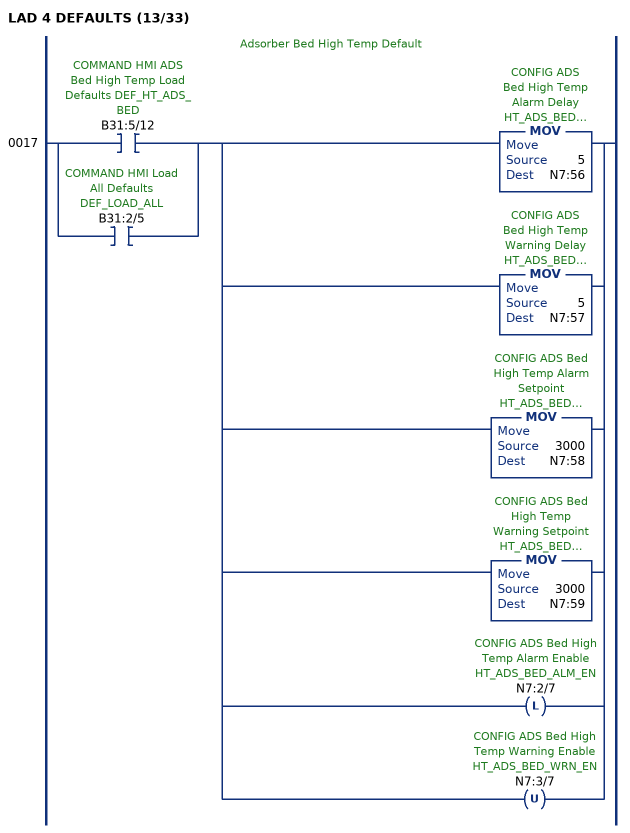
% Rung: 17 %
% Adsorber Bed High Temp Default %
SOR BST XIC B31:5/12 NXB XIC B31:2/5 BND BST MOV 5 N7:56 NXB MOV 5 N7:57 NXB MOV 3000 N7:58 NXB MOV 3000 N7:59 NXB OTL N7:2/7 NXB OTU N7:3/7 BND EOR
%   B31:5/12  DEF_HT_ADS_BED  "COMMAND HMI ADS Bed High Temp Load Defaults" %
%   B31:2/5  DEF_LOAD_ALL  "COMMAND HMI Load All Defaults" %
%   N7:56  HT_ADS_BED_ALM_DLY  "CONFIG ADS Bed High Temp Alarm Delay" %
%   N7:57  HT_ADS_BED_WRN_DLY  "CONFIG ADS Bed High Temp Warning Delay" %
%   N7:58  HT_ADS_BED_ALM_SP  "CONFIG ADS Bed High Temp Alarm Setpoint" %
%   N7:59  HT_ADS_BED_WRN_SP  "CONFIG ADS Bed High Temp Warning Setpoint" %
%   N7:2/7  HT_ADS_BED_ALM_EN  "CONFIG ADS Bed High Temp Alarm Enable" %
%   N7:3/7  HT_ADS_BED_WRN_EN  "CONFIG ADS Bed High Temp Warning Enable" %

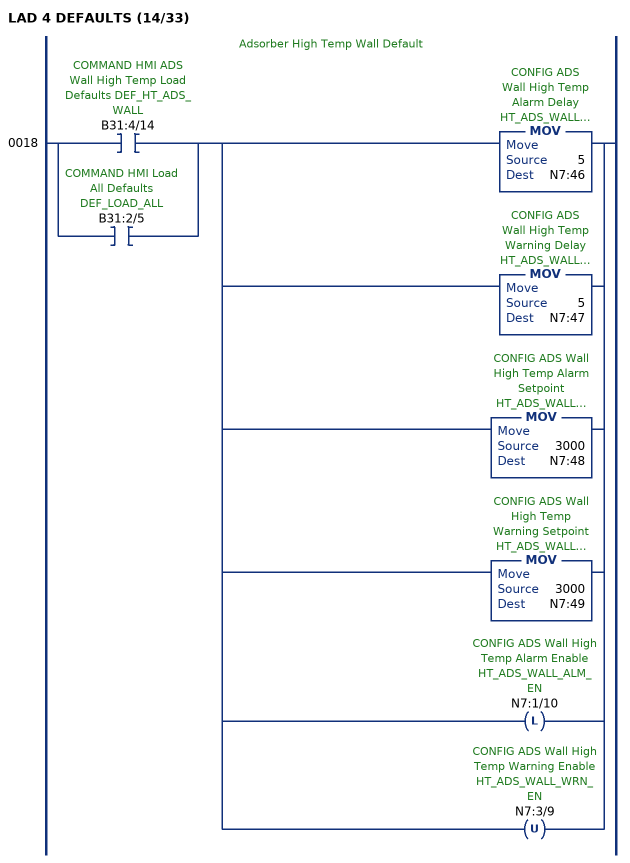
% Rung: 18 %
% Adsorber High Temp Wall Default %
SOR BST XIC B31:4/14 NXB XIC B31:2/5 BND BST MOV 5 N7:46 NXB MOV 5 N7:47 NXB MOV 3000 N7:48 NXB MOV 3000 N7:49 NXB OTL N7:1/10 NXB OTU N7:3/9 BND EOR
%   B31:4/14  DEF_HT_ADS_WALL  "COMMAND HMI ADS Wall High Temp Load Defaults" %
%   B31:2/5  DEF_LOAD_ALL  "COMMAND HMI Load All Defaults" %
%   N7:46  HT_ADS_WALL_ALM_DLY  "CONFIG ADS Wall High Temp Alarm Delay" %
%   N7:47  HT_ADS_WALL_WRN_DLY  "CONFIG ADS Wall High Temp Warning Delay" %
%   N7:48  HT_ADS_WALL_ALM_SP  "CONFIG ADS Wall High Temp Alarm Setpoint" %
%   N7:49  HT_ADS_WALL_WRN_SP  "CONFIG ADS Wall High Temp Warning Setpoint" %
%   N7:1/10  HT_ADS_WALL_ALM_EN  "CONFIG ADS Wall High Temp Alarm Enable" %
%   N7:3/9  HT_ADS_WALL_WRN_EN  "CONFIG ADS Wall High Temp Warning Enable" %

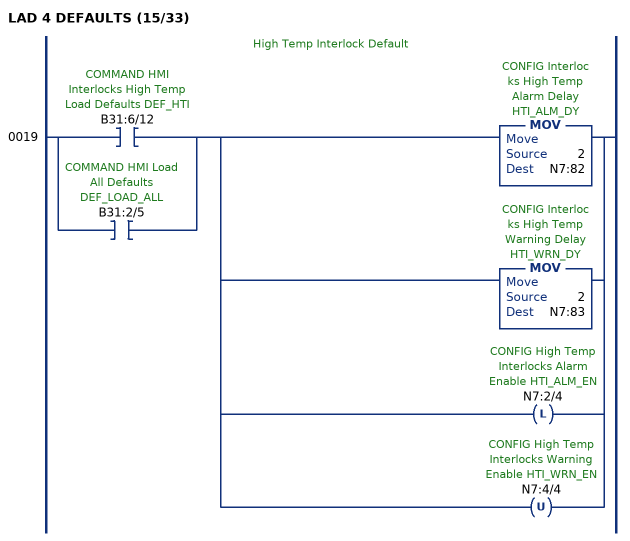
% Rung: 19 %
% High Temp Interlock Default %
SOR BST XIC B31:6/12 NXB XIC B31:2/5 BND BST MOV 2 N7:82 NXB MOV 2 N7:83 NXB OTL N7:2/4 NXB OTU N7:4/4 BND EOR
%   B31:6/12  DEF_HTI  "COMMAND HMI Interlocks High Temp Load Defaults" %
%   B31:2/5  DEF_LOAD_ALL  "COMMAND HMI Load All Defaults" %
%   N7:82  HTI_ALM_DY  "CONFIG Interlocks High Temp Alarm Delay" %
%   N7:83  HTI_WRN_DY  "CONFIG Interlocks High Temp Warning Delay" %
%   N7:2/4  HTI_ALM_EN  "CONFIG High Temp Interlocks Alarm Enable" %
%   N7:4/4  HTI_WRN_EN  "CONFIG High Temp Interlocks Warning Enable" %

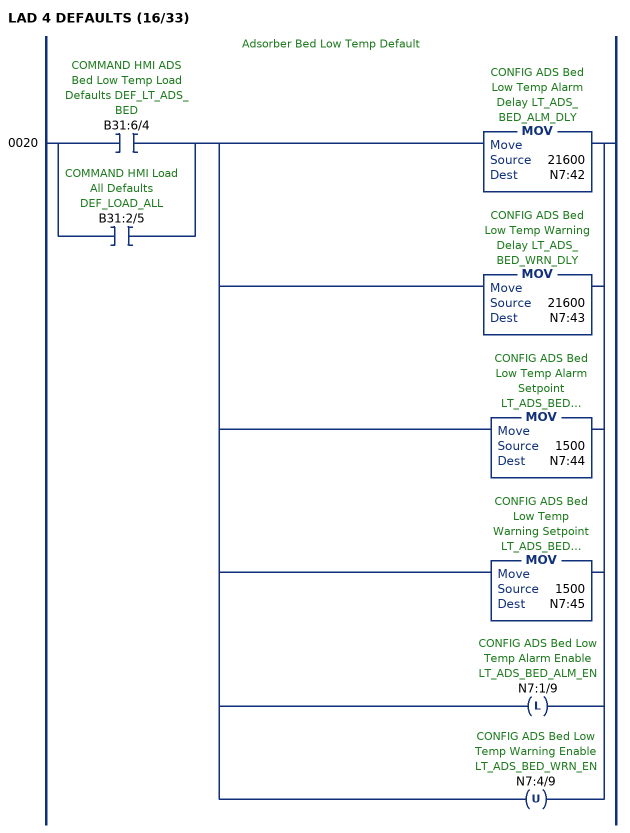
% Rung: 20 %
% Adsorber Bed Low Temp Default %
SOR BST XIC B31:6/4 NXB XIC B31:2/5 BND BST MOV 21600 N7:42 NXB MOV 21600 N7:43 NXB MOV 1500 N7:44 NXB MOV 1500 N7:45 NXB OTL N7:1/9 NXB OTU N7:4/9 BND EOR
%   B31:6/4  DEF_LT_ADS_BED  "COMMAND HMI ADS Bed Low Temp Load Defaults" %
%   B31:2/5  DEF_LOAD_ALL  "COMMAND HMI Load All Defaults" %
%   N7:42  LT_ADS_BED_ALM_DLY  "CONFIG ADS Bed Low Temp Alarm Delay" %
%   N7:43  LT_ADS_BED_WRN_DLY  "CONFIG ADS Bed Low Temp Warning Delay" %
%   N7:44  LT_ADS_BED_ALM_SP  "CONFIG ADS Bed Low Temp Alarm Setpoint" %
%   N7:45  LT_ADS_BED_WRN_SP  "CONFIG ADS Bed Low Temp Warning Setpoint" %
%   N7:1/9  LT_ADS_BED_ALM_EN  "CONFIG ADS Bed Low Temp Alarm Enable" %
%   N7:4/9  LT_ADS_BED_WRN_EN  "CONFIG ADS Bed Low Temp Warning Enable" %

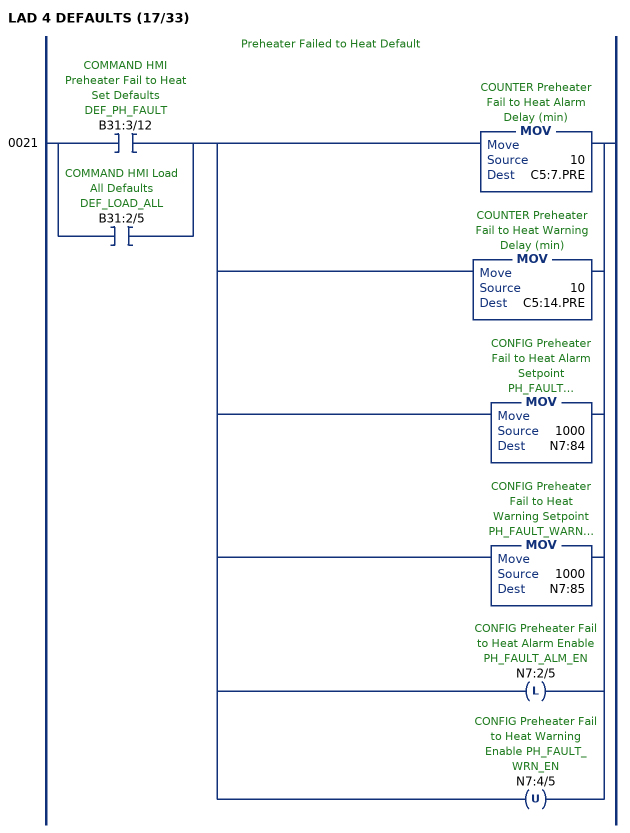
% Rung: 21 %
% Preheater Failed to Heat Default %
SOR BST XIC B31:3/12 NXB XIC B31:2/5 BND BST MOV 10 C5:7.PRE NXB MOV 10 C5:14.PRE NXB MOV 1000 N7:84 NXB MOV 1000 N7:85 NXB OTL N7:2/5 NXB OTU N7:4/5 BND EOR
%   B31:3/12  DEF_PH_FAULT  "COMMAND HMI Preheater Fail to Heat Set Defaults" %
%   B31:2/5  DEF_LOAD_ALL  "COMMAND HMI Load All Defaults" %
%   C5:7.PRE  "COUNTER Preheater Fail to Heat Alarm Delay (min)" %
%   C5:14.PRE  "COUNTER Preheater Fail to Heat Warning Delay (min)" %
%   N7:84  PH_FAULT_ALARM_SP  "CONFIG Preheater Fail to Heat Alarm Setpoint" %
%   N7:85  PH_FAULT_WARN_SP  "CONFIG Preheater Fail to Heat Warning Setpoint" %
%   N7:2/5  PH_FAULT_ALM_EN  "CONFIG Preheater Fail to Heat Alarm Enable" %
%   N7:4/5  PH_FAULT_WRN_EN  "CONFIG Preheater Fail to Heat Warning Enable" %

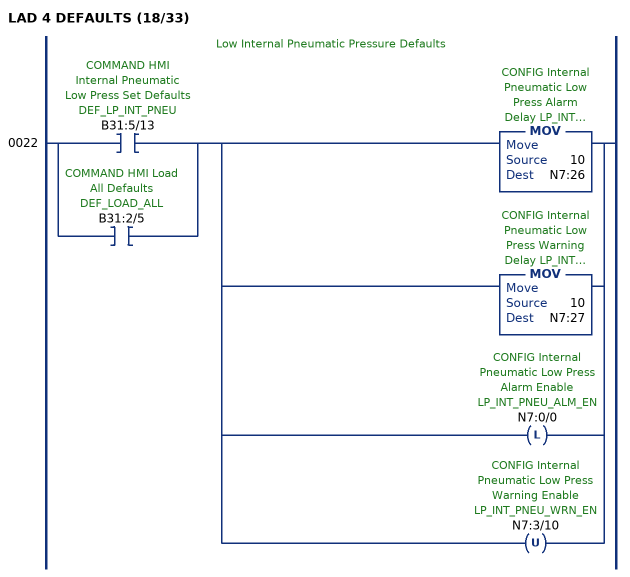
% Rung: 22 %
% Low Internal Pneumatic Pressure Defaults %
SOR BST XIC B31:5/13 NXB XIC B31:2/5 BND BST MOV 10 N7:26 NXB MOV 10 N7:27 NXB OTL N7:0/0 NXB OTU N7:3/10 BND EOR
%   B31:5/13  DEF_LP_INT_PNEU  "COMMAND HMI Internal Pneumatic Low Press Set Defaults" %
%   B31:2/5  DEF_LOAD_ALL  "COMMAND HMI Load All Defaults" %
%   N7:26  LP_INT_PNEU_ALM_DLY  "CONFIG Internal Pneumatic Low Press Alarm Delay" %
%   N7:27  LP_INT_PNEU_WRN_DLY  "CONFIG Internal Pneumatic Low Press Warning Delay" %
%   N7:0/0  LP_INT_PNEU_ALM_EN  "CONFIG Internal Pneumatic Low Press Alarm Enable" %
%   N7:3/10  LP_INT_PNEU_WRN_EN  "CONFIG Internal Pneumatic Low Press Warning Enable" %

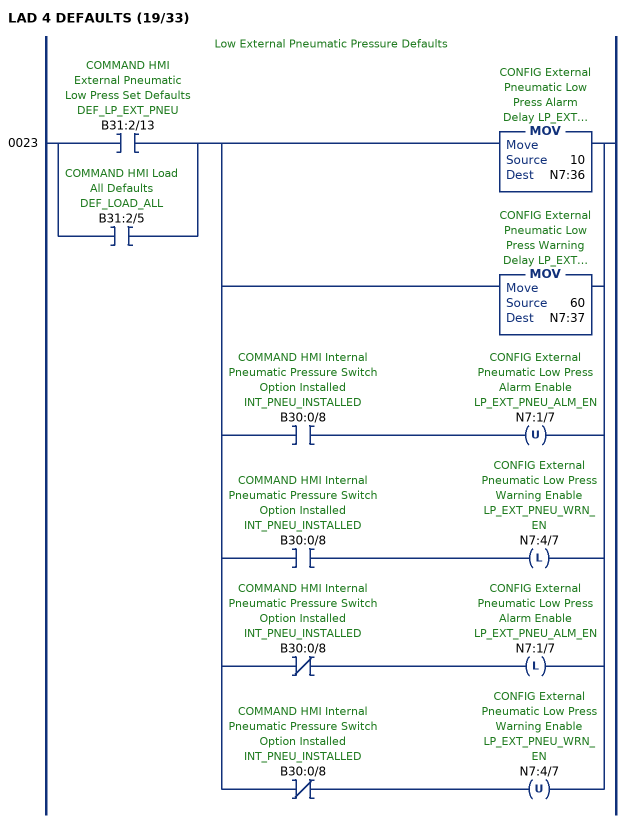
% Rung: 23 %
% Low External Pneumatic Pressure Defaults %
SOR BST XIC B31:2/13 NXB XIC B31:2/5 BND BST MOV 10 N7:36 NXB MOV 60 N7:37 NXB XIC B30:0/8 OTU N7:1/7 NXB XIC B30:0/8 OTL N7:4/7 NXB XIO B30:0/8 OTL N7:1/7 NXB XIO B30:0/8 OTU N7:4/7 BND EOR
%   B31:2/13  DEF_LP_EXT_PNEU  "COMMAND HMI External Pneumatic Low Press Set Defaults" %
%   B31:2/5  DEF_LOAD_ALL  "COMMAND HMI Load All Defaults" %
%   N7:36  LP_EXT_PNEU_ALM_DLY  "CONFIG External Pneumatic Low Press Alarm Delay" %
%   N7:37  LP_EXT_PNEU_WRN_DLY  "CONFIG External Pneumatic Low Press Warning Delay" %
%   B30:0/8  INT_PNEU_INSTALLED  "COMMAND HMI Internal Pneumatic Pressure Switch Option Installed" %
%   N7:1/7  LP_EXT_PNEU_ALM_EN  "CONFIG External Pneumatic Low Press Alarm Enable" %
%   N7:4/7  LP_EXT_PNEU_WRN_EN  "CONFIG External Pneumatic Low Press Warning Enable" %

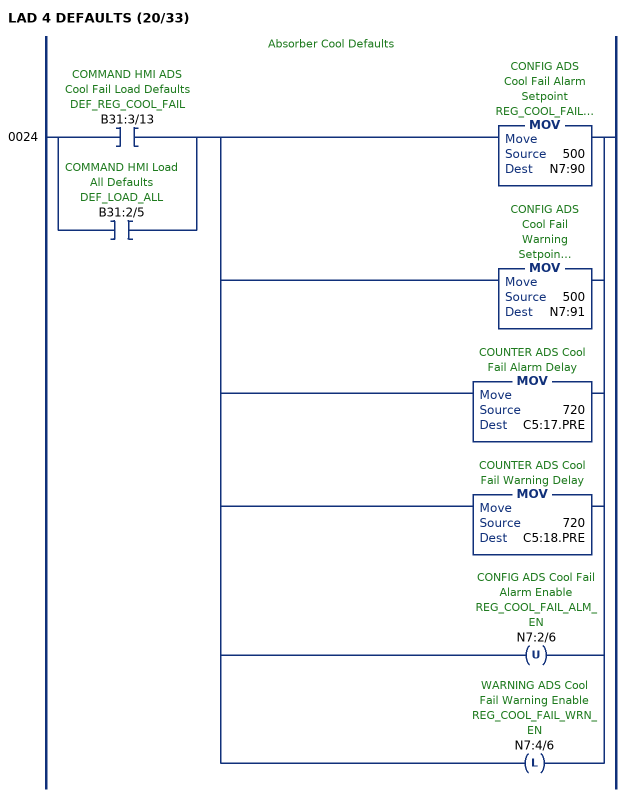
% Rung: 24 %
% Absorber Cool Defaults %
SOR BST XIC B31:3/13 NXB XIC B31:2/5 BND BST MOV 500 N7:90 NXB MOV 500 N7:91 NXB MOV 720 C5:17.PRE NXB MOV 720 C5:18.PRE NXB OTU N7:2/6 NXB OTL N7:4/6 BND EOR
%   B31:3/13  DEF_REG_COOL_FAIL  "COMMAND HMI ADS Cool Fail Load Defaults" %
%   B31:2/5  DEF_LOAD_ALL  "COMMAND HMI Load All Defaults" %
%   N7:90  REG_COOL_FAIL_ALM_SP  "CONFIG ADS Cool Fail Alarm Setpoint" %
%   N7:91  REG_COOL_FAIL_WRN_SP  "CONFIG ADS Cool Fail Warning Setpoint" %
%   C5:17.PRE  "COUNTER ADS Cool Fail Alarm Delay" %
%   C5:18.PRE  "COUNTER ADS Cool Fail Warning Delay" %
%   N7:2/6  REG_COOL_FAIL_ALM_EN  "CONFIG ADS Cool Fail Alarm Enable" %
%   N7:4/6  REG_COOL_FAIL_WRN_EN  "WARNING ADS Cool Fail Warning Enable" %

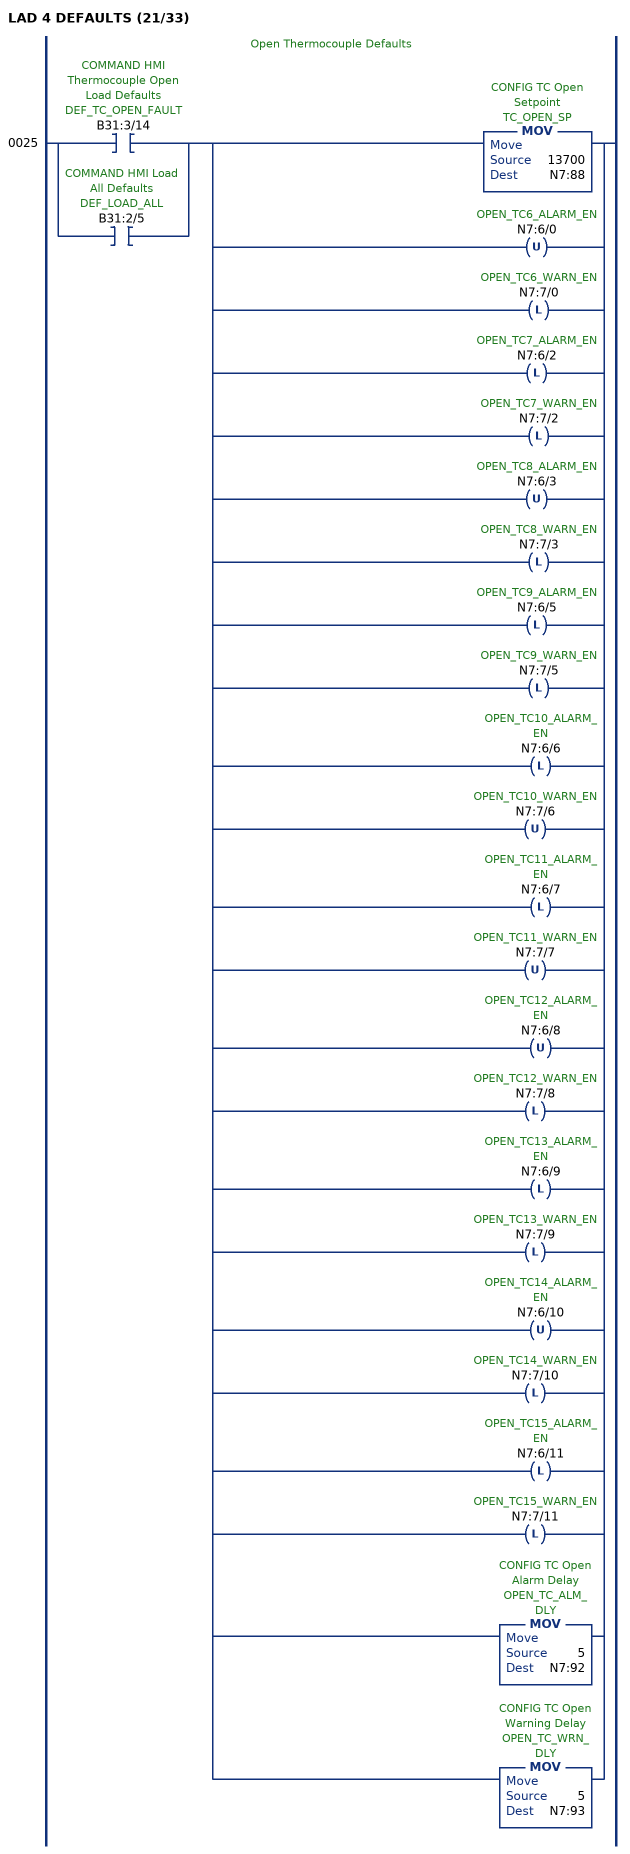
% Rung: 25 %
% Open Thermocouple Defaults %
SOR BST XIC B31:3/14 NXB XIC B31:2/5 BND BST MOV 13700 N7:88 NXB OTU N7:6/0 NXB OTL N7:7/0 NXB OTL N7:6/2 NXB OTL N7:7/2 NXB OTU N7:6/3 NXB OTL N7:7/3 NXB OTL N7:6/5 NXB OTL N7:7/5 NXB OTL N7:6/6 NXB OTU N7:7/6 NXB OTL N7:6/7 NXB OTU N7:7/7 NXB OTU N7:6/8 NXB OTL N7:7/8 NXB OTL N7:6/9 NXB OTL N7:7/9 NXB OTU N7:6/10 NXB OTL N7:7/10 NXB OTL N7:6/11 NXB OTL N7:7/11 NXB MOV 5 N7:92 NXB MOV 5 N7:93 BND EOR
%   B31:3/14  DEF_TC_OPEN_FAULT  "COMMAND HMI Thermocouple Open Load Defaults" %
%   B31:2/5  DEF_LOAD_ALL  "COMMAND HMI Load All Defaults" %
%   N7:88  TC_OPEN_SP  "CONFIG TC Open Setpoint" %
%   N7:6/0  OPEN_TC6_ALARM_EN %
%   N7:7/0  OPEN_TC6_WARN_EN %
%   N7:6/2  OPEN_TC7_ALARM_EN %
%   N7:7/2  OPEN_TC7_WARN_EN %
%   N7:6/3  OPEN_TC8_ALARM_EN %
%   N7:7/3  OPEN_TC8_WARN_EN %
%   N7:6/5  OPEN_TC9_ALARM_EN %
%   N7:7/5  OPEN_TC9_WARN_EN %
%   N7:6/6  OPEN_TC10_ALARM_EN %
%   N7:7/6  OPEN_TC10_WARN_EN %
%   N7:6/7  OPEN_TC11_ALARM_EN %
%   N7:7/7  OPEN_TC11_WARN_EN %
%   N7:6/8  OPEN_TC12_ALARM_EN %
%   N7:7/8  OPEN_TC12_WARN_EN %
%   N7:6/9  OPEN_TC13_ALARM_EN %
%   N7:7/9  OPEN_TC13_WARN_EN %
%   N7:6/10  OPEN_TC14_ALARM_EN %
%   N7:7/10  OPEN_TC14_WARN_EN %
%   N7:6/11  OPEN_TC15_ALARM_EN %
%   N7:7/11  OPEN_TC15_WARN_EN %
%   N7:92  OPEN_TC_ALM_DLY  "CONFIG TC Open Alarm Delay" %
%   N7:93  OPEN_TC_WRN_DLY  "CONFIG TC Open Warning Delay" %

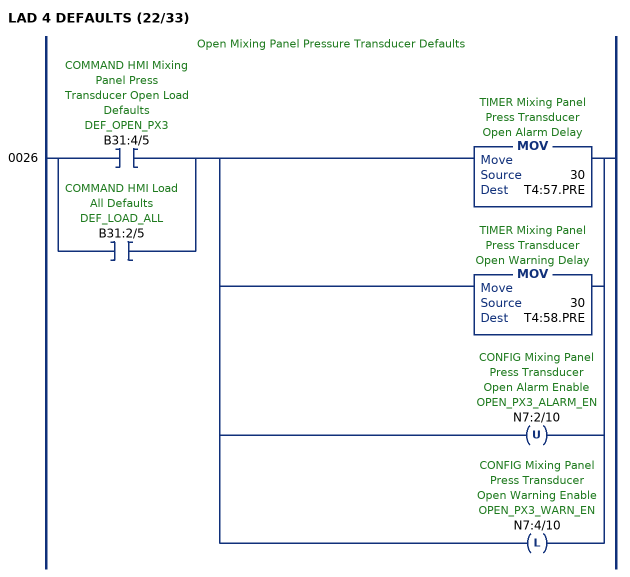
% Rung: 26 %
% Open Mixing Panel Pressure Transducer Defaults %
SOR BST XIC B31:4/5 NXB XIC B31:2/5 BND BST MOV 30 T4:57.PRE NXB MOV 30 T4:58.PRE NXB OTU N7:2/10 NXB OTL N7:4/10 BND EOR
%   B31:4/5  DEF_OPEN_PX3  "COMMAND HMI Mixing Panel Press Transducer Open Load Defaults" %
%   B31:2/5  DEF_LOAD_ALL  "COMMAND HMI Load All Defaults" %
%   T4:57.PRE  "TIMER Mixing Panel Press Transducer Open Alarm Delay" %
%   T4:58.PRE  "TIMER Mixing Panel Press Transducer Open Warning Delay" %
%   N7:2/10  OPEN_PX3_ALARM_EN  "CONFIG Mixing Panel Press Transducer Open Alarm Enable" %
%   N7:4/10  OPEN_PX3_WARN_EN  "CONFIG Mixing Panel Press Transducer Open Warning Enable" %

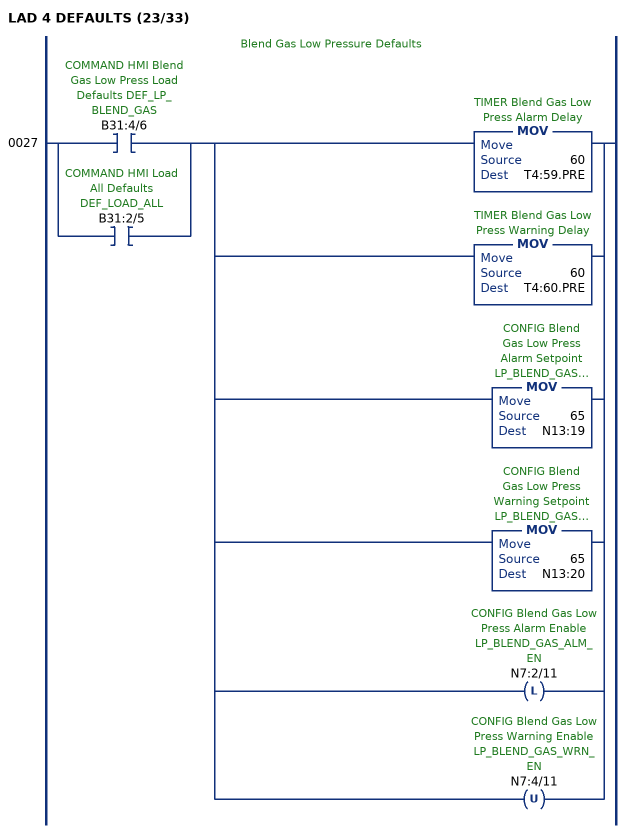
% Rung: 27 %
% Blend Gas Low Pressure Defaults %
SOR BST XIC B31:4/6 NXB XIC B31:2/5 BND BST MOV 60 T4:59.PRE NXB MOV 60 T4:60.PRE NXB MOV 65 N13:19 NXB MOV 65 N13:20 NXB OTL N7:2/11 NXB OTU N7:4/11 BND EOR
%   B31:4/6  DEF_LP_BLEND_GAS  "COMMAND HMI Blend Gas Low Press Load Defaults" %
%   B31:2/5  DEF_LOAD_ALL  "COMMAND HMI Load All Defaults" %
%   T4:59.PRE  "TIMER Blend Gas Low Press Alarm Delay" %
%   T4:60.PRE  "TIMER Blend Gas Low Press Warning Delay" %
%   N13:19  LP_BLEND_GAS_ALM_SP  "CONFIG Blend Gas Low Press Alarm Setpoint" %
%   N13:20  LP_BLEND_GAS_WRN_SP  "CONFIG Blend Gas Low Press Warning Setpoint" %
%   N7:2/11  LP_BLEND_GAS_ALM_EN  "CONFIG Blend Gas Low Press Alarm Enable" %
%   N7:4/11  LP_BLEND_GAS_WRN_EN  "CONFIG Blend Gas Low Press Warning Enable" %

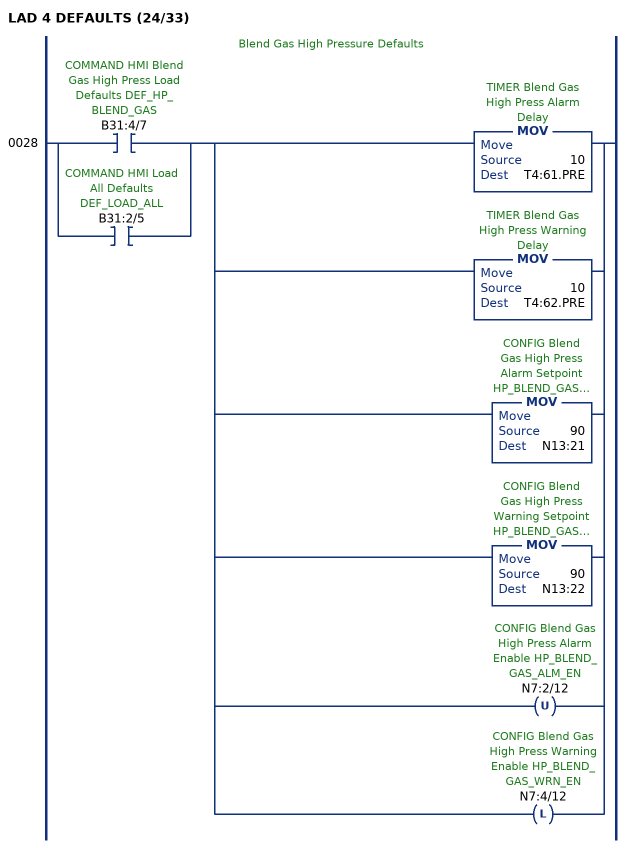
% Rung: 28 %
% Blend Gas High Pressure Defaults %
SOR BST XIC B31:4/7 NXB XIC B31:2/5 BND BST MOV 10 T4:61.PRE NXB MOV 10 T4:62.PRE NXB MOV 90 N13:21 NXB MOV 90 N13:22 NXB OTU N7:2/12 NXB OTL N7:4/12 BND EOR
%   B31:4/7  DEF_HP_BLEND_GAS  "COMMAND HMI Blend Gas High Press Load Defaults" %
%   B31:2/5  DEF_LOAD_ALL  "COMMAND HMI Load All Defaults" %
%   T4:61.PRE  "TIMER Blend Gas High Press Alarm Delay" %
%   T4:62.PRE  "TIMER Blend Gas High Press Warning Delay" %
%   N13:21  HP_BLEND_GAS_ALM_SP  "CONFIG Blend Gas High Press Alarm Setpoint" %
%   N13:22  HP_BLEND_GAS_WRN_SP  "CONFIG Blend Gas High Press Warning Setpoint" %
%   N7:2/12  HP_BLEND_GAS_ALM_EN  "CONFIG Blend Gas High Press Alarm Enable" %
%   N7:4/12  HP_BLEND_GAS_WRN_EN  "CONFIG Blend Gas High Press Warning Enable" %

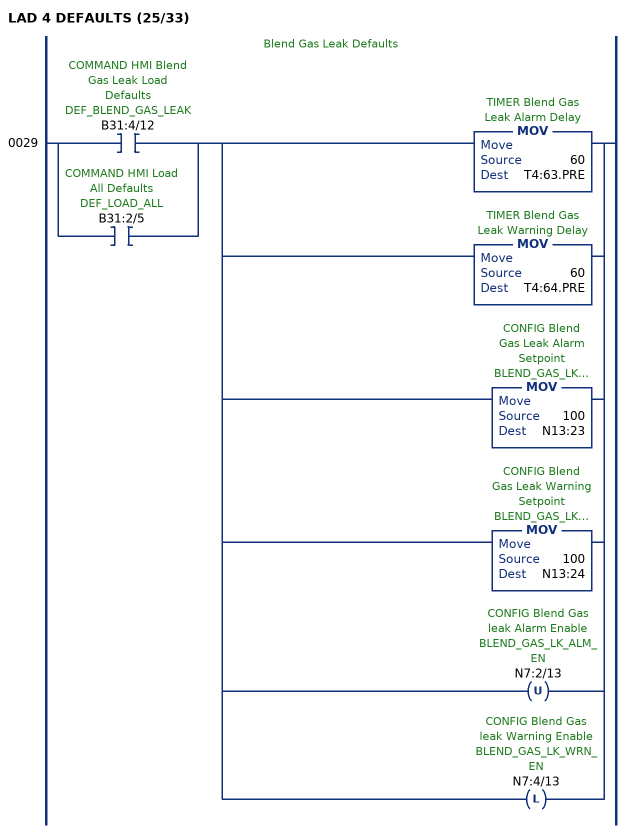
% Rung: 29 %
% Blend Gas Leak Defaults %
SOR BST XIC B31:4/12 NXB XIC B31:2/5 BND BST MOV 60 T4:63.PRE NXB MOV 60 T4:64.PRE NXB MOV 100 N13:23 NXB MOV 100 N13:24 NXB OTU N7:2/13 NXB OTL N7:4/13 BND EOR
%   B31:4/12  DEF_BLEND_GAS_LEAK  "COMMAND HMI Blend Gas Leak Load Defaults" %
%   B31:2/5  DEF_LOAD_ALL  "COMMAND HMI Load All Defaults" %
%   T4:63.PRE  "TIMER Blend Gas Leak Alarm Delay" %
%   T4:64.PRE  "TIMER Blend Gas Leak Warning Delay" %
%   N13:23  BLEND_GAS_LK_ALM_SP  "CONFIG Blend Gas Leak Alarm Setpoint" %
%   N13:24  BLEND_GAS_LK_WRN_SP  "CONFIG Blend Gas Leak Warning Setpoint" %
%   N7:2/13  BLEND_GAS_LK_ALM_EN  "CONFIG Blend Gas leak Alarm Enable" %
%   N7:4/13  BLEND_GAS_LK_WRN_EN  "CONFIG Blend Gas leak Warning Enable" %

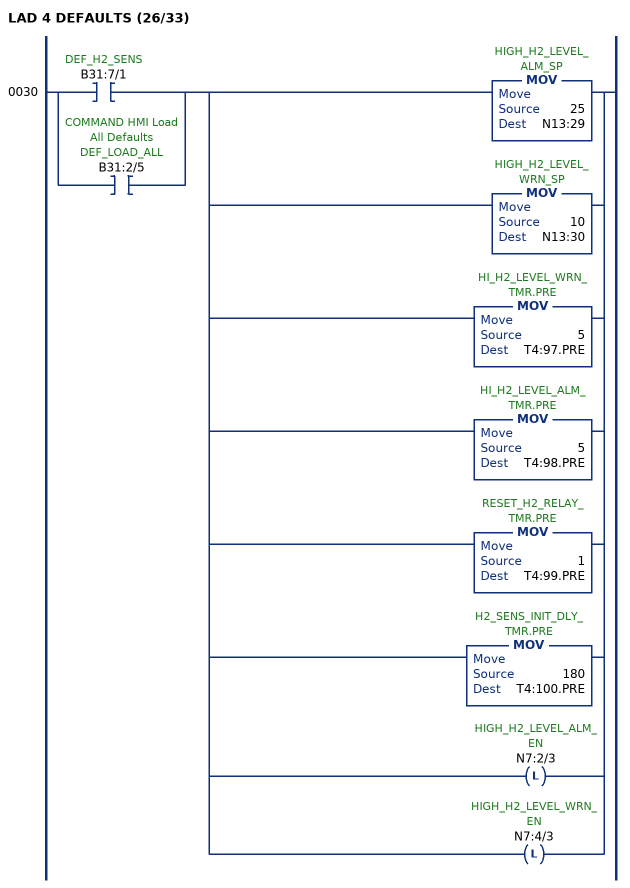
% Rung: 30 %
SOR BST XIC B31:7/1 NXB XIC B31:2/5 BND BST MOV 25 N13:29 NXB MOV 10 N13:30 NXB MOV 5 T4:97.PRE NXB MOV 5 T4:98.PRE NXB MOV 1 T4:99.PRE NXB MOV 180 T4:100.PRE NXB OTL N7:2/3 NXB OTL N7:4/3 BND EOR
%   B31:7/1  DEF_H2_SENS %
%   B31:2/5  DEF_LOAD_ALL  "COMMAND HMI Load All Defaults" %
%   N13:29  HIGH_H2_LEVEL_ALM_SP %
%   N13:30  HIGH_H2_LEVEL_WRN_SP %
%   T4:97  HI_H2_LEVEL_WRN_TMR %
%   T4:98  HI_H2_LEVEL_ALM_TMR %
%   T4:99  RESET_H2_RELAY_TMR %
%   T4:100  H2_SENS_INIT_DLY_TMR %
%   N7:2/3  HIGH_H2_LEVEL_ALM_EN %
%   N7:4/3  HIGH_H2_LEVEL_WRN_EN %

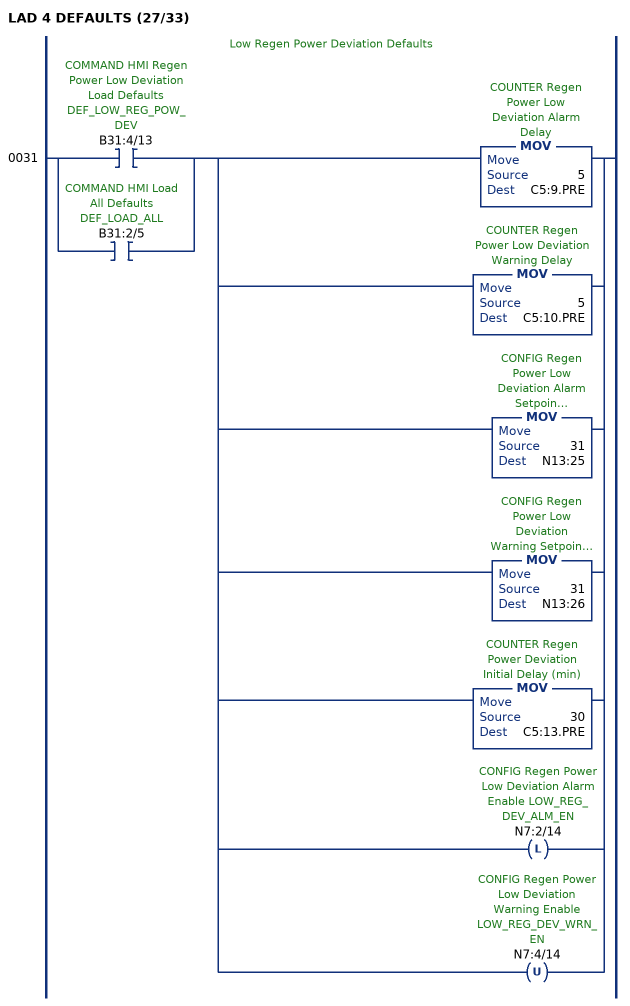
% Rung: 31 %
% Low Regen Power Deviation Defaults %
SOR BST XIC B31:4/13 NXB XIC B31:2/5 BND BST MOV 5 C5:9.PRE NXB MOV 5 C5:10.PRE NXB MOV 31 N13:25 NXB MOV 31 N13:26 NXB MOV 30 C5:13.PRE NXB OTL N7:2/14 NXB OTU N7:4/14 BND EOR
%   B31:4/13  DEF_LOW_REG_POW_DEV  "COMMAND HMI Regen Power Low Deviation Load Defaults" %
%   B31:2/5  DEF_LOAD_ALL  "COMMAND HMI Load All Defaults" %
%   C5:9.PRE  "COUNTER Regen Power Low Deviation Alarm Delay" %
%   C5:10.PRE  "COUNTER Regen Power Low Deviation Warning Delay" %
%   N13:25  LOW_REG_DEV_ALM_SP  "CONFIG Regen Power Low Deviation Alarm Setpoint" %
%   N13:26  LOW_REG_DEV_WRN_SP  "CONFIG Regen Power Low Deviation Warning Setpoint" %
%   C5:13.PRE  "COUNTER Regen Power Deviation Initial Delay (min)" %
%   N7:2/14  LOW_REG_DEV_ALM_EN  "CONFIG Regen Power Low Deviation Alarm Enable" %
%   N7:4/14  LOW_REG_DEV_WRN_EN  "CONFIG Regen Power Low Deviation Warning Enable" %

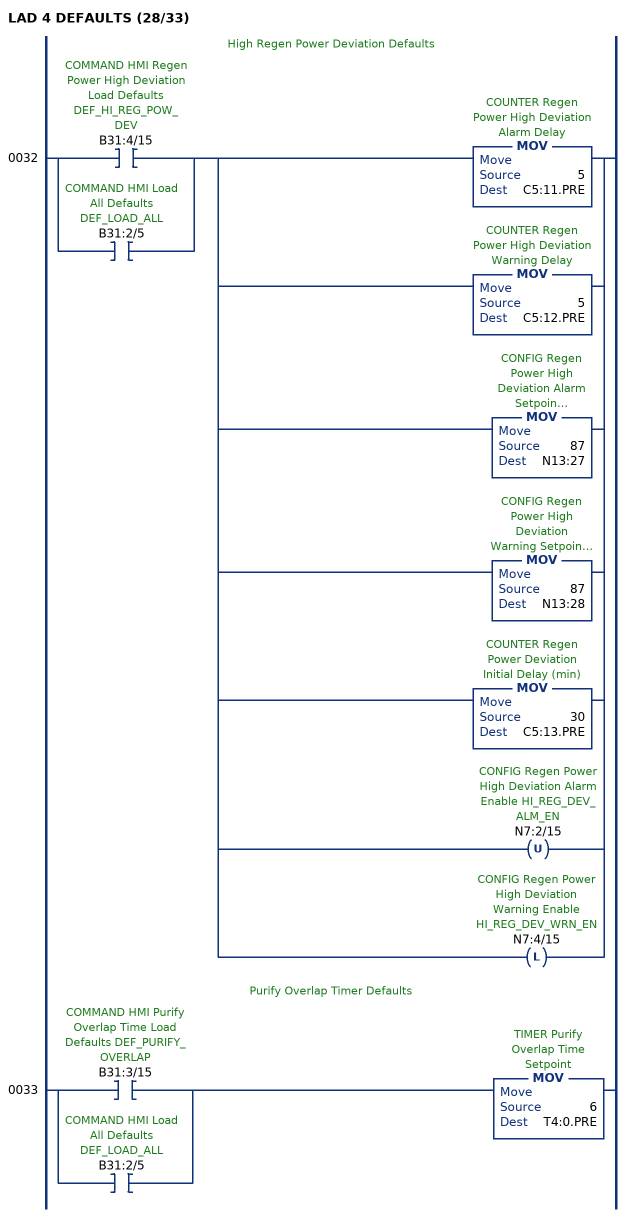
% Rung: 32 %
% High Regen Power Deviation Defaults %
SOR BST XIC B31:4/15 NXB XIC B31:2/5 BND BST MOV 5 C5:11.PRE NXB MOV 5 C5:12.PRE NXB MOV 87 N13:27 NXB MOV 87 N13:28 NXB MOV 30 C5:13.PRE NXB OTU N7:2/15 NXB OTL N7:4/15 BND EOR
%   B31:4/15  DEF_HI_REG_POW_DEV  "COMMAND HMI Regen Power High Deviation Load Defaults" %
%   B31:2/5  DEF_LOAD_ALL  "COMMAND HMI Load All Defaults" %
%   C5:11.PRE  "COUNTER Regen Power High Deviation Alarm Delay" %
%   C5:12.PRE  "COUNTER Regen Power High Deviation Warning Delay" %
%   N13:27  HI_REG_DEV_ALM_SP  "CONFIG Regen Power High Deviation Alarm Setpoint" %
%   N13:28  HI_REG_DEV_WRN_SP  "CONFIG Regen Power High Deviation Warning Setpoint" %
%   C5:13.PRE  "COUNTER Regen Power Deviation Initial Delay (min)" %
%   N7:2/15  HI_REG_DEV_ALM_EN  "CONFIG Regen Power High Deviation Alarm Enable" %
%   N7:4/15  HI_REG_DEV_WRN_EN  "CONFIG Regen Power High Deviation Warning Enable" %
% Rung: 33 %
% Purify Overlap Timer Defaults %
SOR BST XIC B31:3/15 NXB XIC B31:2/5 BND MOV 6 T4:0.PRE EOR
%   B31:3/15  DEF_PURIFY_OVERLAP  "COMMAND HMI Purify Overlap Time Load Defaults" %
%   B31:2/5  DEF_LOAD_ALL  "COMMAND HMI Load All Defaults" %
%   T4:0.PRE  "TIMER Purify Overlap Time Setpoint" %

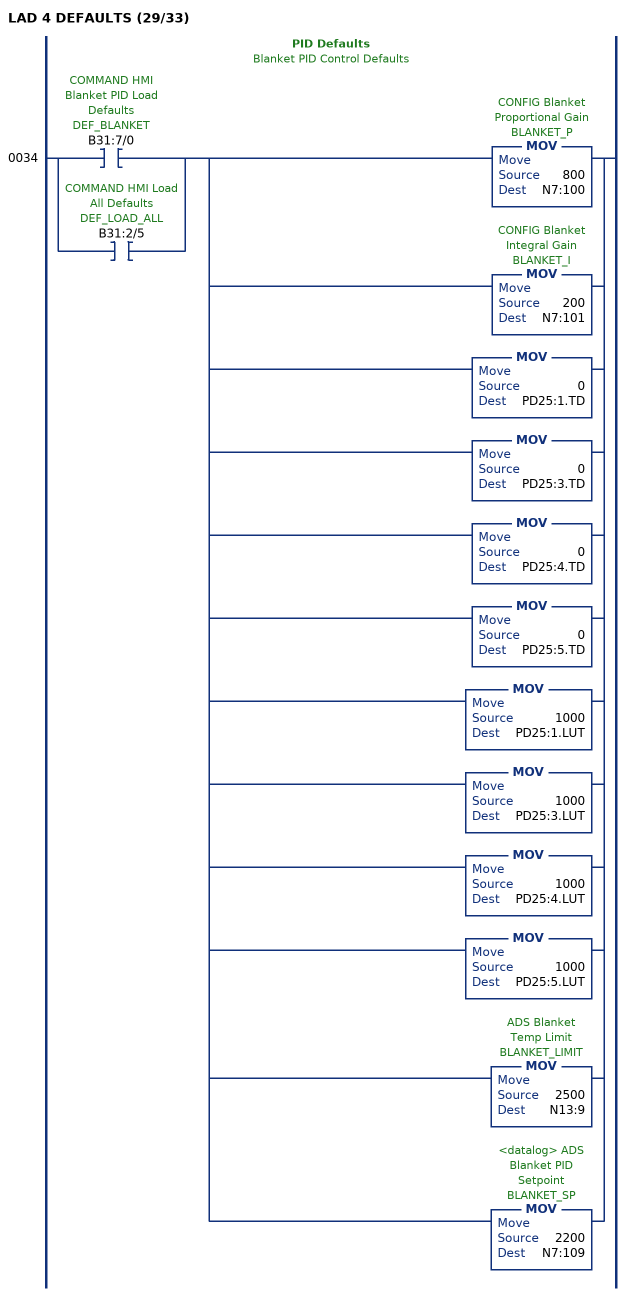
% Rung: 34 %
% TITLE: PID Defaults %
% Blanket PID Control Defaults %
SOR BST XIC B31:7/0 NXB XIC B31:2/5 BND BST MOV 800 N7:100 NXB MOV 200 N7:101 NXB MOV 0 PD25:1.TD NXB MOV 0 PD25:3.TD NXB MOV 0 PD25:4.TD NXB MOV 0 PD25:5.TD NXB MOV 1000 PD25:1.LUT NXB MOV 1000 PD25:3.LUT NXB MOV 1000 PD25:4.LUT NXB MOV 1000 PD25:5.LUT NXB MOV 2500 N13:9 NXB MOV 2200 N7:109 BND EOR
%   B31:7/0  DEF_BLANKET  "COMMAND HMI Blanket PID Load Defaults" %
%   B31:2/5  DEF_LOAD_ALL  "COMMAND HMI Load All Defaults" %
%   N7:100  BLANKET_P  "CONFIG Blanket Proportional Gain" %
%   N7:101  BLANKET_I  "CONFIG Blanket Integral Gain" %
%   N13:9  BLANKET_LIMIT  "ADS Blanket Temp Limit" %
%   N7:109  BLANKET_SP  "<datalog> ADS Blanket PID Setpoint" %

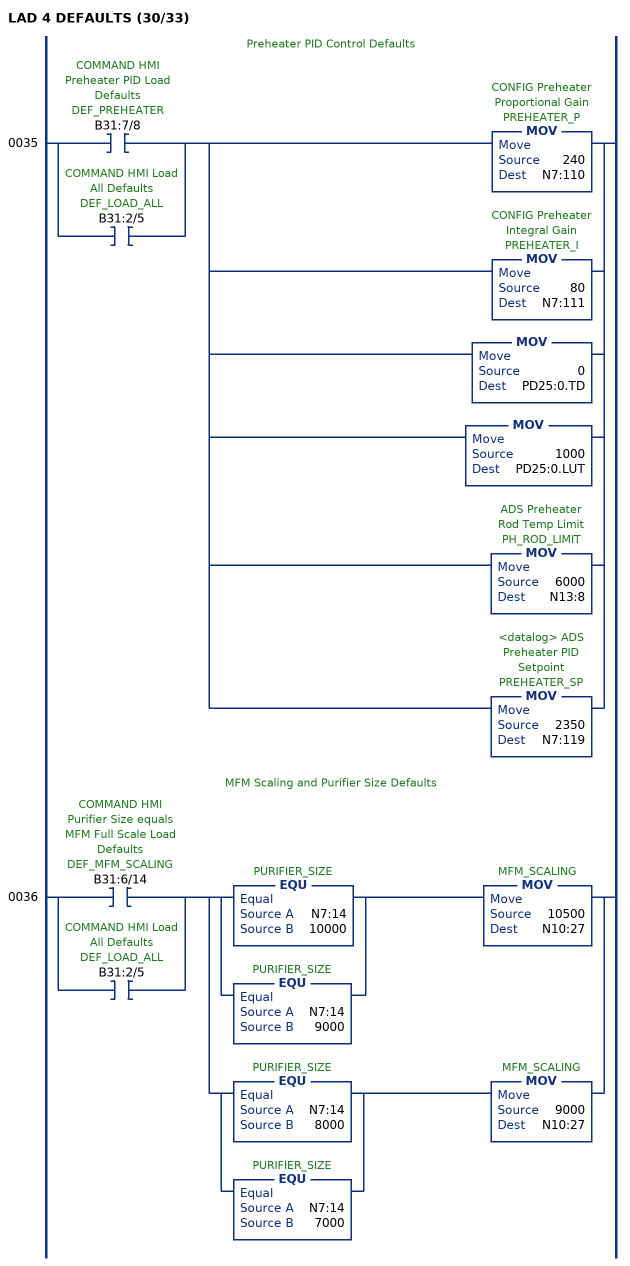
% Rung: 35 %
% Preheater PID Control Defaults %
SOR BST XIC B31:7/8 NXB XIC B31:2/5 BND BST MOV 240 N7:110 NXB MOV 80 N7:111 NXB MOV 0 PD25:0.TD NXB MOV 1000 PD25:0.LUT NXB MOV 6000 N13:8 NXB MOV 2350 N7:119 BND EOR
%   B31:7/8  DEF_PREHEATER  "COMMAND HMI Preheater PID Load Defaults" %
%   B31:2/5  DEF_LOAD_ALL  "COMMAND HMI Load All Defaults" %
%   N7:110  PREHEATER_P  "CONFIG Preheater Proportional Gain" %
%   N7:111  PREHEATER_I  "CONFIG Preheater Integral Gain" %
%   N13:8  PH_ROD_LIMIT  "ADS Preheater Rod Temp Limit" %
%   N7:119  PREHEATER_SP  "<datalog> ADS Preheater PID Setpoint" %
% Rung: 36 %
% MFM Scaling and Purifier Size Defaults %
SOR BST XIC B31:6/14 NXB XIC B31:2/5 BND BST BST EQU N7:14 10000 NXB EQU N7:14 9000 BND MOV 10500 N10:27 NXB BST EQU N7:14 8000 NXB EQU N7:14 7000 BND MOV 9000 N10:27 BND EOR
%   B31:6/14  DEF_MFM_SCALING  "COMMAND HMI Purifier Size equals MFM Full Scale Load Defaults" %
%   B31:2/5  DEF_LOAD_ALL  "COMMAND HMI Load All Defaults" %
%   N7:14  PURIFIER_SIZE %
%   N10:27  MFM_SCALING %

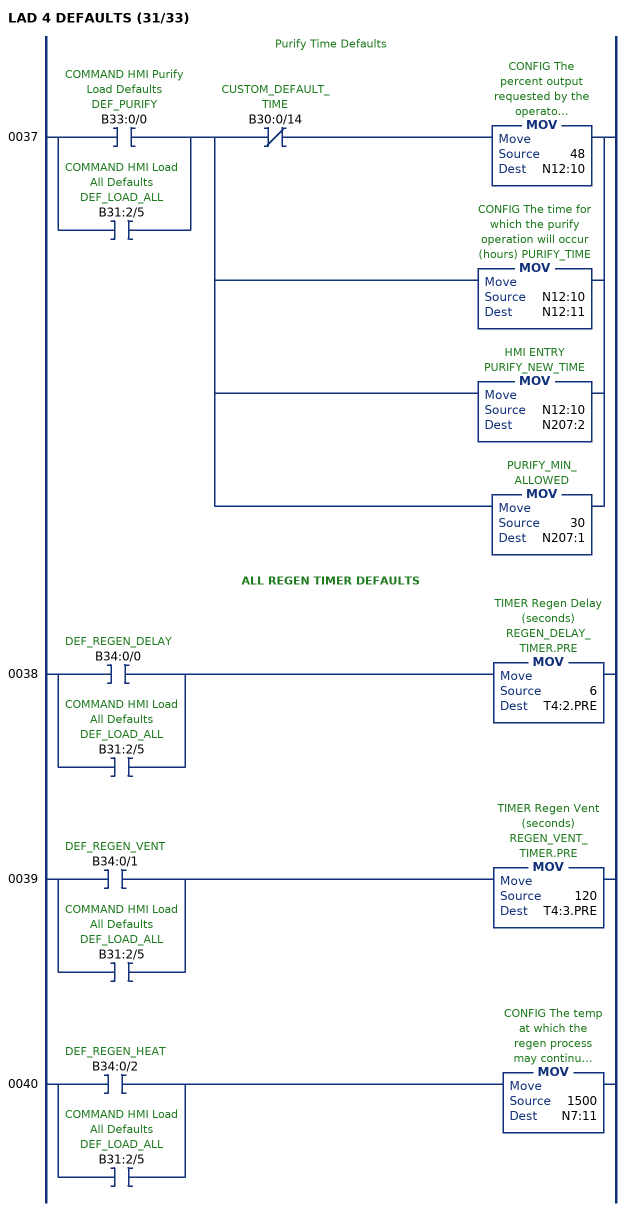
% Rung: 37 %
% Purify Time Defaults %
SOR BST XIC B33:0/0 NXB XIC B31:2/5 BND BST XIO B30:0/14 MOV 48 N12:10 NXB MOV N12:10 N12:11 NXB MOV N12:10 N207:2 NXB MOV 30 N207:1 BND EOR
%   B33:0/0  DEF_PURIFY  "COMMAND HMI Purify Load Defaults" %
%   B31:2/5  DEF_LOAD_ALL  "COMMAND HMI Load All Defaults" %
%   B30:0/14  CUSTOM_DEFAULT_TIME %
%   N12:10  DEFAULT_PURIFY_TIME  "CONFIG The percent output requested by the operator (percent)" %
%   N12:11  PURIFY_TIME  "CONFIG The time for which the purify operation will occur (hours)" %
%   N207:2  PURIFY_NEW_TIME  "HMI ENTRY" %
%   N207:1  PURIFY_MIN_ALLOWED %
% Rung: 38 %
% TITLE: ALL REGEN TIMER DEFAULTS %
SOR BST XIC B34:0/0 NXB XIC B31:2/5 BND MOV 6 T4:2.PRE EOR
%   B34:0/0  DEF_REGEN_DELAY %
%   B31:2/5  DEF_LOAD_ALL  "COMMAND HMI Load All Defaults" %
%   T4:2  REGEN_DELAY_TIMER  "TIMER Regen Delay (seconds)" %
% Rung: 39 %
SOR BST XIC B34:0/1 NXB XIC B31:2/5 BND MOV 120 T4:3.PRE EOR
%   B34:0/1  DEF_REGEN_VENT %
%   B31:2/5  DEF_LOAD_ALL  "COMMAND HMI Load All Defaults" %
%   T4:3  REGEN_VENT_TIMER  "TIMER Regen Vent (seconds)" %
% Rung: 40 %
SOR BST XIC B34:0/2 NXB XIC B31:2/5 BND MOV 1500 N7:11 EOR
%   B34:0/2  DEF_REGEN_HEAT %
%   B31:2/5  DEF_LOAD_ALL  "COMMAND HMI Load All Defaults" %
%   N7:11  ADS_BED_TEMP_HIGH  "CONFIG The temp at which the regen process may continue" %

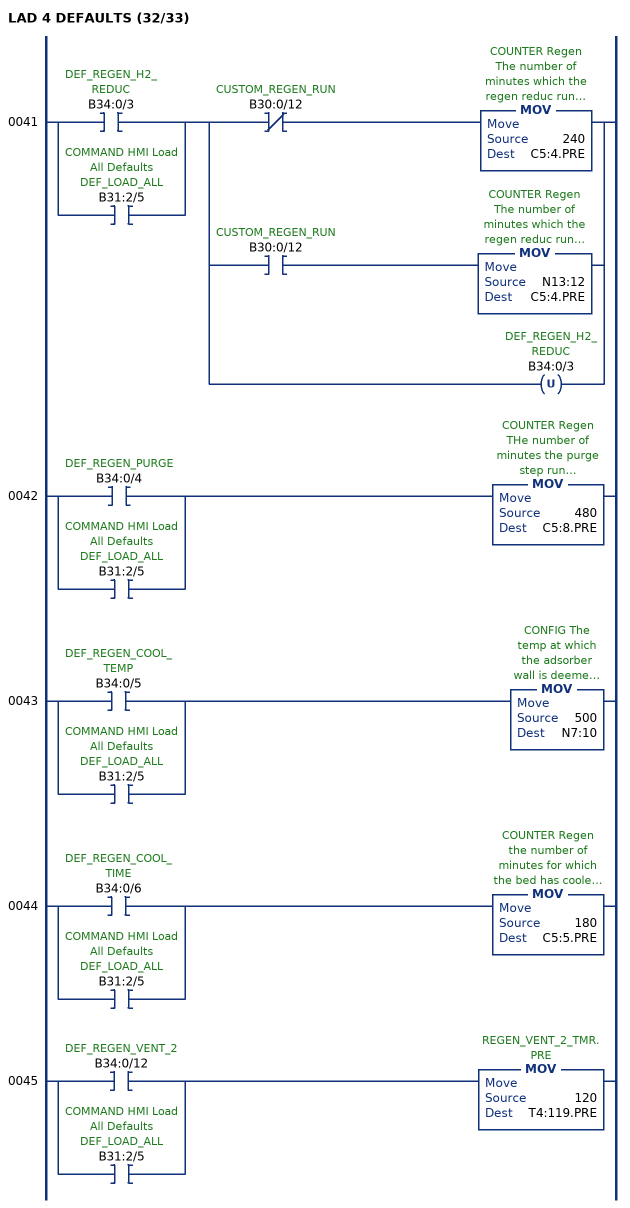
% Rung: 41 %
SOR BST XIC B34:0/3 NXB XIC B31:2/5 BND BST XIO B30:0/12 MOV 240 C5:4.PRE NXB XIC B30:0/12 MOV N13:12 C5:4.PRE NXB OTU B34:0/3 BND EOR
%   B34:0/3  DEF_REGEN_H2_REDUC %
%   B31:2/5  DEF_LOAD_ALL  "COMMAND HMI Load All Defaults" %
%   B30:0/12  CUSTOM_REGEN_RUN %
%   C5:4  REGEN_REDUC_MINUTE  "COUNTER Regen The number of minutes which the regen reduc runs" %
%   N13:12  NEW_REGEN_RUN_TIME %
% Rung: 42 %
SOR BST XIC B34:0/4 NXB XIC B31:2/5 BND MOV 480 C5:8.PRE EOR
%   B34:0/4  DEF_REGEN_PURGE %
%   B31:2/5  DEF_LOAD_ALL  "COMMAND HMI Load All Defaults" %
%   C5:8  REGEN_PURGE_MINUTES  "COUNTER Regen THe number of minutes the purge step runs" %
% Rung: 43 %
SOR BST XIC B34:0/5 NXB XIC B31:2/5 BND MOV 500 N7:10 EOR
%   B34:0/5  DEF_REGEN_COOL_TEMP %
%   B31:2/5  DEF_LOAD_ALL  "COMMAND HMI Load All Defaults" %
%   N7:10  ADS_WALL_TEMP_COOL  "CONFIG The temp at which the adsorber wall is deemed to be cool enough to purify" %
% Rung: 44 %
SOR BST XIC B34:0/6 NXB XIC B31:2/5 BND MOV 180 C5:5.PRE EOR
%   B34:0/6  DEF_REGEN_COOL_TIME %
%   B31:2/5  DEF_LOAD_ALL  "COMMAND HMI Load All Defaults" %
%   C5:5  REGEN_COOL_MINUTE  "COUNTER Regen the number of minutes for which the bed has cooled" %
% Rung: 45 %
SOR BST XIC B34:0/12 NXB XIC B31:2/5 BND MOV 120 T4:119.PRE EOR
%   B34:0/12  DEF_REGEN_VENT_2 %
%   B31:2/5  DEF_LOAD_ALL  "COMMAND HMI Load All Defaults" %
%   T4:119  REGEN_VENT_2_TMR %

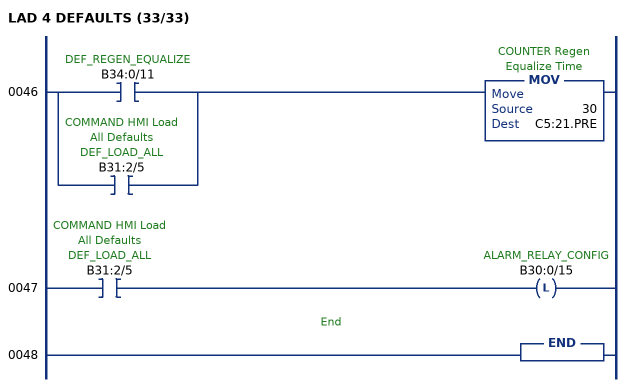
% Rung: 46 %
SOR BST XIC B34:0/11 NXB XIC B31:2/5 BND MOV 30 C5:21.PRE EOR
%   B34:0/11  DEF_REGEN_EQUALIZE %
%   B31:2/5  DEF_LOAD_ALL  "COMMAND HMI Load All Defaults" %
%   C5:21.PRE  "COUNTER Regen Equalize Time" %
% Rung: 47 %
SOR XIC B31:2/5 OTL B30:0/15 EOR
%   B31:2/5  DEF_LOAD_ALL  "COMMAND HMI Load All Defaults" %
%   B30:0/15  ALARM_RELAY_CONFIG %
% Rung: 48 %
% End %
SOR END EOR

LADDER 5 "SYS_FAULTS"    % Monitors the system fault conditions %
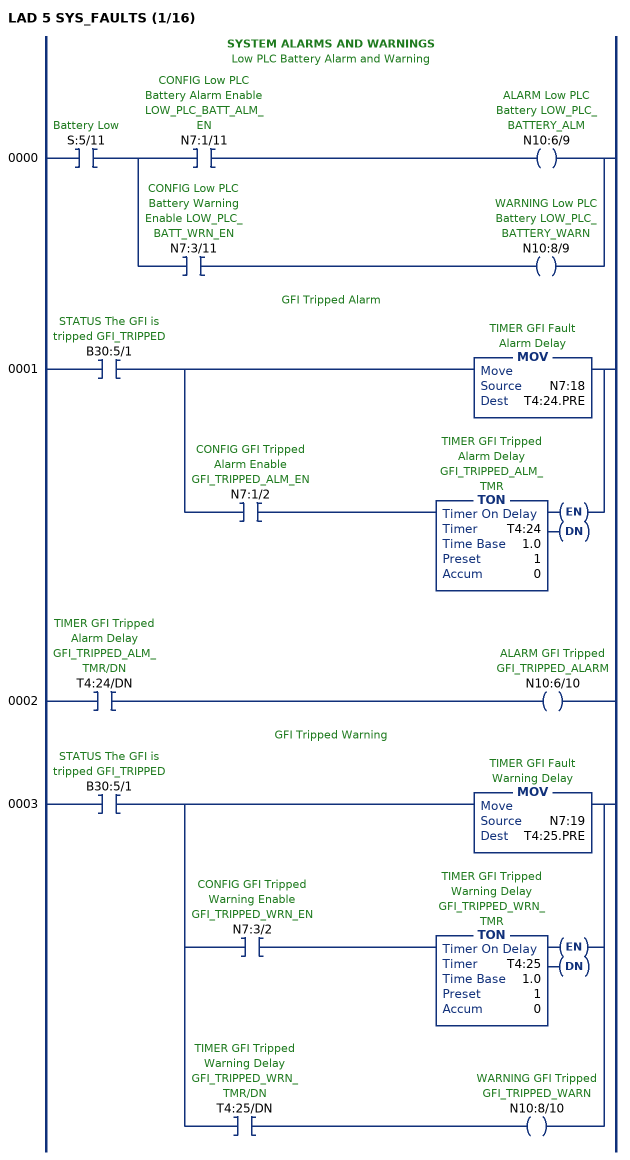
% Rung: 0 %
% TITLE: SYSTEM ALARMS AND WARNINGS %
% Low PLC Battery Alarm and Warning %
SOR XIC S:5/11 BST XIC N7:1/11 OTE N10:6/9 NXB XIC N7:3/11 OTE N10:8/9 BND EOR
%   S:5/11  "Battery Low" %
%   N7:1/11  LOW_PLC_BATT_ALM_EN  "CONFIG Low PLC Battery Alarm Enable" %
%   N10:6/9  LOW_PLC_BATTERY_ALM  "ALARM Low PLC Battery" %
%   N7:3/11  LOW_PLC_BATT_WRN_EN  "CONFIG Low PLC Battery Warning Enable" %
%   N10:8/9  LOW_PLC_BATTERY_WARN  "WARNING Low PLC Battery" %
% Rung: 1 %
% GFI Tripped Alarm %
SOR XIC B30:5/1 BST MOV N7:18 T4:24.PRE NXB XIC N7:1/2 TON T4:24 1.0 1 0 BND EOR
%   B30:5/1  GFI_TRIPPED  "STATUS The GFI is tripped" %
%   N7:18  GFI_TRIPPED_ALM_DLY  "CONFIG GFI Fault Alarm Delay" %
%   T4:24.PRE  "TIMER GFI Fault Alarm Delay" %
%   N7:1/2  GFI_TRIPPED_ALM_EN  "CONFIG GFI Tripped Alarm Enable" %
%   T4:24  GFI_TRIPPED_ALM_TMR  "TIMER GFI Tripped Alarm Delay" %
% Rung: 2 %
SOR XIC T4:24/DN OTE N10:6/10 EOR
%   T4:24  GFI_TRIPPED_ALM_TMR  "TIMER GFI Tripped Alarm Delay" %
%   N10:6/10  GFI_TRIPPED_ALARM  "ALARM GFI Tripped" %
% Rung: 3 %
% GFI Tripped Warning %
SOR XIC B30:5/1 BST MOV N7:19 T4:25.PRE NXB XIC N7:3/2 TON T4:25 1.0 1 0 NXB XIC T4:25/DN OTE N10:8/10 BND EOR
%   B30:5/1  GFI_TRIPPED  "STATUS The GFI is tripped" %
%   N7:19  GFI_TRIPPED_WRN_DLY  "CONFIG GFI Fault Warning Delay" %
%   T4:25.PRE  "TIMER GFI Fault Warning Delay" %
%   N7:3/2  GFI_TRIPPED_WRN_EN  "CONFIG GFI Tripped Warning Enable" %
%   T4:25  GFI_TRIPPED_WRN_TMR  "TIMER GFI Tripped Warning Delay" %
%   N10:8/10  GFI_TRIPPED_WARN  "WARNING GFI Tripped" %

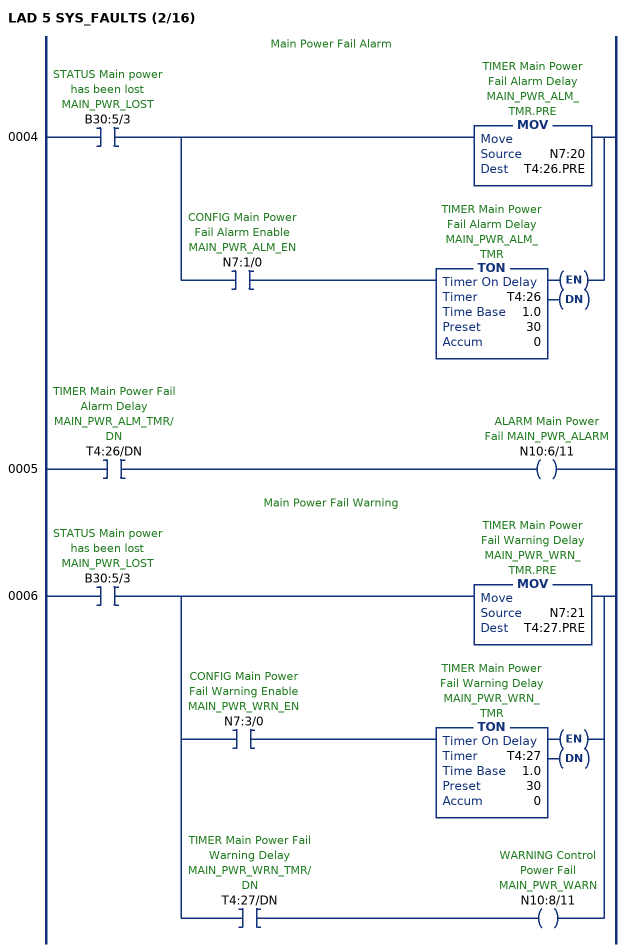
% Rung: 4 %
% Main Power Fail Alarm %
SOR XIC B30:5/3 BST MOV N7:20 T4:26.PRE NXB XIC N7:1/0 TON T4:26 1.0 30 0 BND EOR
%   B30:5/3  MAIN_PWR_LOST  "STATUS Main power has been lost" %
%   N7:20  PWR_FAIL_ALM_DELAY  "CONFIG Main Power Fail Alarm Delay" %
%   T4:26  MAIN_PWR_ALM_TMR  "TIMER Main Power Fail Alarm Delay" %
%   N7:1/0  MAIN_PWR_ALM_EN  "CONFIG Main Power Fail Alarm Enable" %
% Rung: 5 %
SOR XIC T4:26/DN OTE N10:6/11 EOR
%   T4:26  MAIN_PWR_ALM_TMR  "TIMER Main Power Fail Alarm Delay" %
%   N10:6/11  MAIN_PWR_ALARM  "ALARM Main Power Fail" %
% Rung: 6 %
% Main Power Fail Warning %
SOR XIC B30:5/3 BST MOV N7:21 T4:27.PRE NXB XIC N7:3/0 TON T4:27 1.0 30 0 NXB XIC T4:27/DN OTE N10:8/11 BND EOR
%   B30:5/3  MAIN_PWR_LOST  "STATUS Main power has been lost" %
%   N7:21  PWR_FAIL_WRN_DELAY  "CONFIG Main Power Fail Warning Delay" %
%   T4:27  MAIN_PWR_WRN_TMR  "TIMER Main Power Fail Warning Delay" %
%   N7:3/0  MAIN_PWR_WRN_EN  "CONFIG Main Power Fail Warning Enable" %
%   N10:8/11  MAIN_PWR_WARN  "WARNING Control Power Fail" %

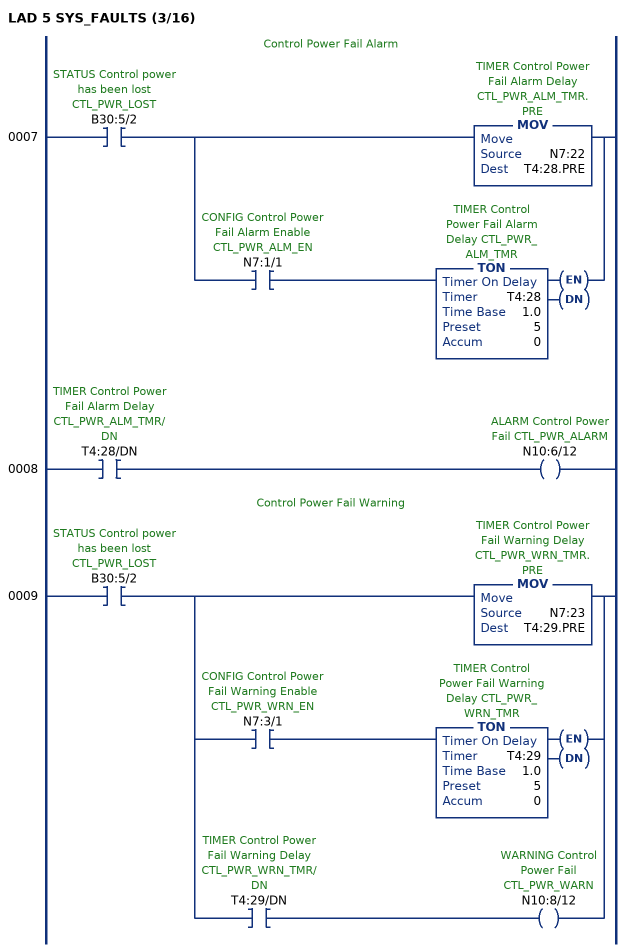
% Rung: 7 %
% Control Power Fail Alarm %
SOR XIC B30:5/2 BST MOV N7:22 T4:28.PRE NXB XIC N7:1/1 TON T4:28 1.0 5 0 BND EOR
%   B30:5/2  CTL_PWR_LOST  "STATUS Control power has been lost" %
%   N7:22  CTL_PWR_FAIL_ALM_DLY  "CONFIG Control Power Fail Alarm Delay" %
%   T4:28  CTL_PWR_ALM_TMR  "TIMER Control Power Fail Alarm Delay" %
%   N7:1/1  CTL_PWR_ALM_EN  "CONFIG Control Power Fail Alarm Enable" %
% Rung: 8 %
SOR XIC T4:28/DN OTE N10:6/12 EOR
%   T4:28  CTL_PWR_ALM_TMR  "TIMER Control Power Fail Alarm Delay" %
%   N10:6/12  CTL_PWR_ALARM  "ALARM Control Power Fail" %
% Rung: 9 %
% Control Power Fail Warning %
SOR XIC B30:5/2 BST MOV N7:23 T4:29.PRE NXB XIC N7:3/1 TON T4:29 1.0 5 0 NXB XIC T4:29/DN OTE N10:8/12 BND EOR
%   B30:5/2  CTL_PWR_LOST  "STATUS Control power has been lost" %
%   N7:23  CTL_PWR_FAIL_WRN_DLY  "CONFIG Control Power Fail Warning Delay" %
%   T4:29  CTL_PWR_WRN_TMR  "TIMER Control Power Fail Warning Delay" %
%   N7:3/1  CTL_PWR_WRN_EN  "CONFIG Control Power Fail Warning Enable" %
%   N10:8/12  CTL_PWR_WARN  "WARNING Control Power Fail" %

